// TIA Portal V20 export
TYPE "LAxisCtrl_typeHoming"
TITLE = LAxisCtrl_typeHoming
// Support: tech.team.motioncontrol@siemens.com 
// Fax: +49 (0) 9131/98-1297
   STRUCT
      position : LReal := 0.0;   // The specified value is used according to the selected "Mode"
      mode : Int := 0;   // Operation mode; 0: Direct homing (absolute); 1:Direct homing (relative); 2:Passive homing (without reset); 3:Active homing; 5:Active homing (Position parameter has no effect); 6:Absolute encoder adjustment (relative); 7:Absolute encoder adjustment (absolute); 8:Passive homing ; 9:Abort passive homing; 10: Passive homing (Position parameter has no effect)
      extendedMode : DInt := -1;   // -1: No extended homing mode (parameter "mode" is effective); 0: Homing on fixed stop;
      extendedModeTorqueLimit : LReal := 0.0;   // Value of the torque/force for extended homing mode
   END_STRUCT;
END_TYPE
